// Base interface for immutable collections
INTERFACE I_Immutable_Collection EXTENDS I_Collection

END_INTERFACE

(* stored: Version 1.1.0.1, ProductVersion 3.1.4024.4
   Itf I_Immutable_Collection: Id {83371683-5a8c-08cf-245b-1b6708129727} *)
